(* Logix 5000 project; controller Sucrose_Main Emulate 5570 rev 20.12; software revision 20.01; part 21 of 30 *)
(* tags used below, declared in another part *)
   CIPRemote : Area_Program;
   FV140501_AOI : QSI_Flow_Valve;   // FV-14-05-01 PRE FILTER TRAIN 1 SUPPLY VALVE
   FV140502_AOI : QSI_Flow_Valve;   // FV-14-05-02 FINAL FILTER TRAIN 1 SUPPLY VALVE
   FV140503_AOI : QSI_Flow_Valve;   // FV-14-05-03 HOT WATER LOW POINT DRAIN VALVE
   FV140601_AOI : QSI_Flow_Valve;   // FV-14-06-01 PRE FILTER TRAIN 2 SUPPLY VALVE
   FV140602_AOI : QSI_Flow_Valve;   // FV-14-06-02 FINAL FILTER TRAIN 2 SUPPLY VALVE
   FV150501_AOI : QSI_Flow_Valve;   // FV-15-05-01 DIVERT TO SCRAP OR TO DRAIN VALVE
   FV230500_AOI : QSI_Flow_Valve;   // FV-23-05-00 SUCROSE LOW POINT DRAIN VALVE
   FV230501_AOI : QSI_Flow_Valve;   // FV-23-05-01-O PRE FILTER TRAIN 1 INLET VALVE OPEN
   FV230502_AOI : QSI_Flow_Valve;   // FV-23-05-02 PRE FILTER TRAIN 1 INLET LOW POINT DRAIN VALVE
   FV230503_AOI : QSI_Flow_Valve;   // FV-23-05-03 PRE FILTER TRAIN 1 INLET LOW POINT DRAIN VALVE
   FV230504_AOI : QSI_Flow_Valve;   // FV-23-05-04 PRE FILTER TRAIN 1 OUTLET LOW POINT DRAIN VALVE
   FV230505_AOI : QSI_Flow_Valve;   // FV-23-05-05 PRE FILTER TRAIN 1 OUTLET LOW POINT DRAIN VALVE
   FV230506_AOI : QSI_Flow_Valve;   // FV-23-05-06-O PRE FILTER TRAIN 1 OUTLET VALVE OPEN
   FV230508_AOI : QSI_Flow_Valve;   // FV-23-05-08-O FINAL FILTER TRAIN 1 INLET VALVE OPEN
   FV230509_AOI : QSI_Flow_Valve;   // FV-23-05-09 FINAL FILTER TRAIN 1 INLET LOW POINT DRAIN VALVE
   FV230510_AOI : QSI_Flow_Valve;   // FV-23-05-10 FINAL FILTER TRAIN 1 INLET LOW POINT DRAIN VALVE
   FV230511_AOI : QSI_Flow_Valve;   // FV-23-05-11 FINAL FILTER TRAIN 1 OUTLET LOW POINT DRAIN VALVE
   FV230512_AOI : QSI_Flow_Valve;   // FV-23-05-12 FINAL FILTER TRAIN 1 OUTLET LOW POINT DRAIN VALVE
   FV230513_AOI : QSI_Flow_Valve;   // FV-23-05-13-O FINAL FILTER TRAIN 1 OUTLET VALVE OPEN
   FV230601_AOI : QSI_Flow_Valve;   // FV-23-06-01-O PRE FILTER TRAIN 2 INLET VALVE OPEN
   FV230602_AOI : QSI_Flow_Valve;   // FV-23-06-02 PRE FILTER TRAIN 2 INLET LOW POINT DRAIN VALVE
   FV230603_AOI : QSI_Flow_Valve;   // FV-23-06-03 PRE FILTER TRAIN 2 INLET LOW POINT DRAIN VALVE
   FV230604_AOI : QSI_Flow_Valve;   // FV-23-06-04 PRE FILTER TRAIN 2 OUTLET LOW POINT DRAIN VALVE
   FV230605_AOI : QSI_Flow_Valve;   // FV-23-06-05 PRE FILTER TRAIN 2 OUTLET LOW POINT DRAIN VALVE
   FV230606_AOI : QSI_Flow_Valve;   // FV-23-06-06-O PRE FILTER TRAIN 2 OUTLET VALVE OPEN
   FV230607_AOI : QSI_Flow_Valve;   // FV-23-06-07 LOW POINT DRAIN VALVE
   FV230608_AOI : QSI_Flow_Valve;   // FV-23-06-08-O FINAL FILTER TRAIN 2 INLET VALVE OPEN
   FV230609_AOI : QSI_Flow_Valve;   // FV-23-06-09 FINAL FILTER TRAIN 2 INLET LOW POINT DRAIN VALVE
   FV230610_AOI : QSI_Flow_Valve;   // FV-23-06-10 FINAL FILTER TRAIN 2 INLET LOW POINT DRAIN VALVE
   FV230611_AOI : QSI_Flow_Valve;   // FV-23-06-11 FINAL FILTER TRAIN 2 OUTLET LOW POINT DRAIN VALVE
   FV230612_AOI : QSI_Flow_Valve;   // FV-23-06-12 FINAL FILTER TRAIN 2 OUTLET LOW POINT DRAIN VALVE
   FV230613_AOI : QSI_Flow_Valve;   // FV-23-06-13-O FINAL FILTER TRAIN 2 OUTLET VALVE OPEN
   ONESHOTBITS : INT[10];
   Rung_Comment : BOOL;
   SECURITY : User_Login;
   SucroseCIP_FILTRATION_REMOTE : CIP_REMOTE;
   SucroseCIP_RUNNING : BOOL;
   SucroseCIP_TK230101_REMOTE : CIP_REMOTE;
   SucroseCIP_TK230201_REMOTE : CIP_REMOTE;
   SucroseCIP_TK230301_REMOTE : CIP_REMOTE;
   SucroseFiltration : Area_Program;
(* Master_Main, continued *)

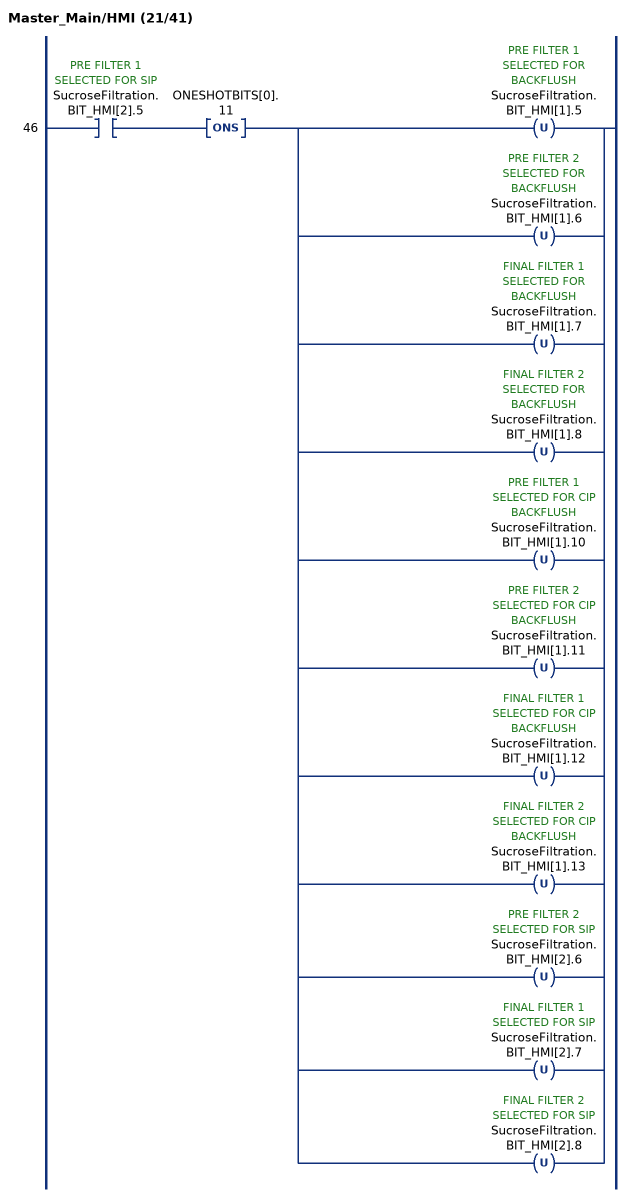
   46: XIC(SucroseFiltration.BIT_HMI[2].5)ONS(ONESHOTBITS[0].11)[OTU(SucroseFiltration.BIT_HMI[1].5) ,OTU(SucroseFiltration.BIT_HMI[1].6) ,OTU(SucroseFiltration.BIT_HMI[1].7) ,OTU(SucroseFiltration.BIT_HMI[1].8) ,OTU(SucroseFiltration.BIT_HMI[1].10) ,OTU(SucroseFiltration.BIT_HMI[1].11) ,OTU(SucroseFiltration.BIT_HMI[1].12) ,OTU(SucroseFiltration.BIT_HMI[1].13) ,OTU(SucroseFiltration.BIT_HMI[2].6) ,OTU(SucroseFiltration.BIT_HMI[2].7) ,OTU(SucroseFiltration.BIT_HMI[2].8) ];
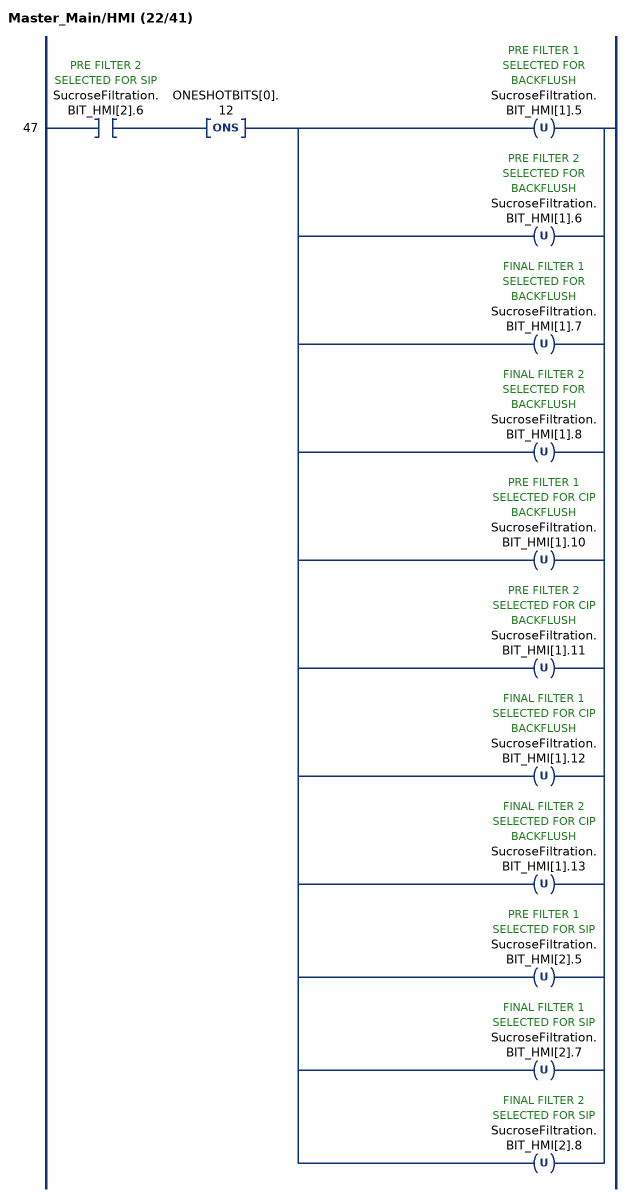
   47: XIC(SucroseFiltration.BIT_HMI[2].6)ONS(ONESHOTBITS[0].12)[OTU(SucroseFiltration.BIT_HMI[1].5) ,OTU(SucroseFiltration.BIT_HMI[1].6) ,OTU(SucroseFiltration.BIT_HMI[1].7) ,OTU(SucroseFiltration.BIT_HMI[1].8) ,OTU(SucroseFiltration.BIT_HMI[1].10) ,OTU(SucroseFiltration.BIT_HMI[1].11) ,OTU(SucroseFiltration.BIT_HMI[1].12) ,OTU(SucroseFiltration.BIT_HMI[1].13) ,OTU(SucroseFiltration.BIT_HMI[2].5) ,OTU(SucroseFiltration.BIT_HMI[2].7) ,OTU(SucroseFiltration.BIT_HMI[2].8) ];
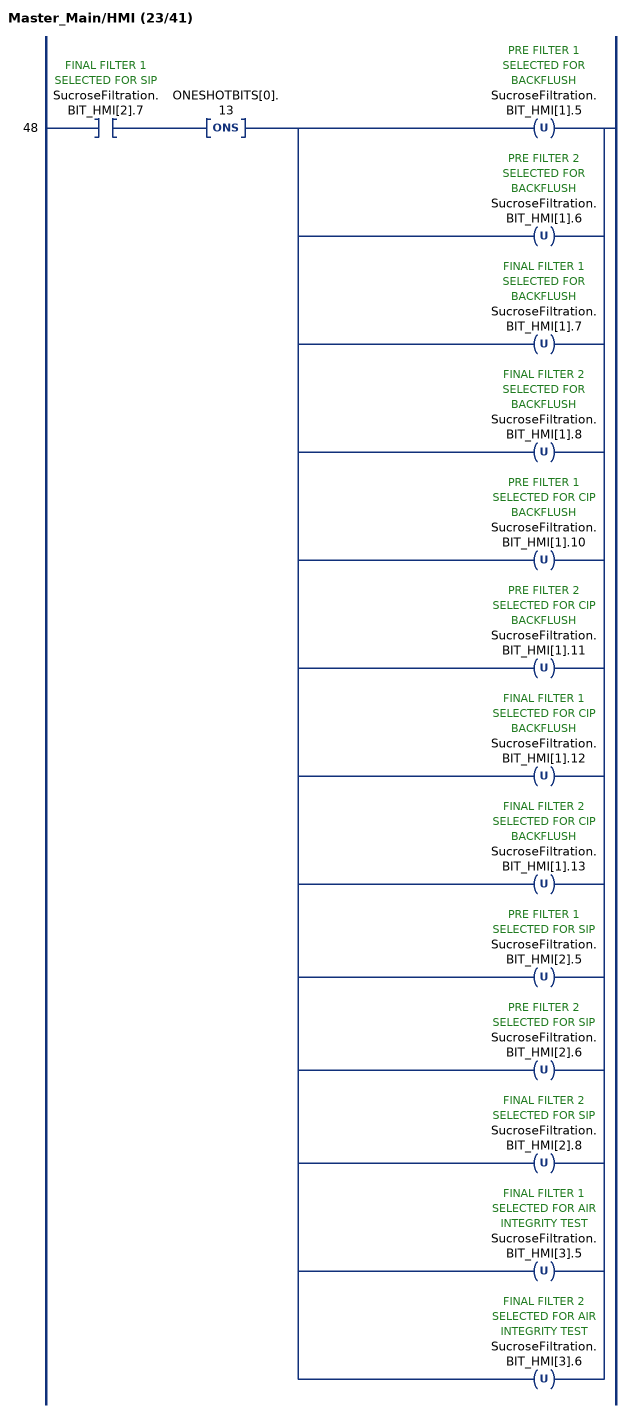
   48: XIC(SucroseFiltration.BIT_HMI[2].7)ONS(ONESHOTBITS[0].13)[OTU(SucroseFiltration.BIT_HMI[1].5) ,OTU(SucroseFiltration.BIT_HMI[1].6) ,OTU(SucroseFiltration.BIT_HMI[1].7) ,OTU(SucroseFiltration.BIT_HMI[1].8) ,OTU(SucroseFiltration.BIT_HMI[1].10) ,OTU(SucroseFiltration.BIT_HMI[1].11) ,OTU(SucroseFiltration.BIT_HMI[1].12) ,OTU(SucroseFiltration.BIT_HMI[1].13) ,OTU(SucroseFiltration.BIT_HMI[2].5) ,OTU(SucroseFiltration.BIT_HMI[2].6) ,OTU(SucroseFiltration.BIT_HMI[2].8) ,OTU(SucroseFiltration.BIT_HMI[3].5) ,OTU(SucroseFiltration.BIT_HMI[3].6) ];
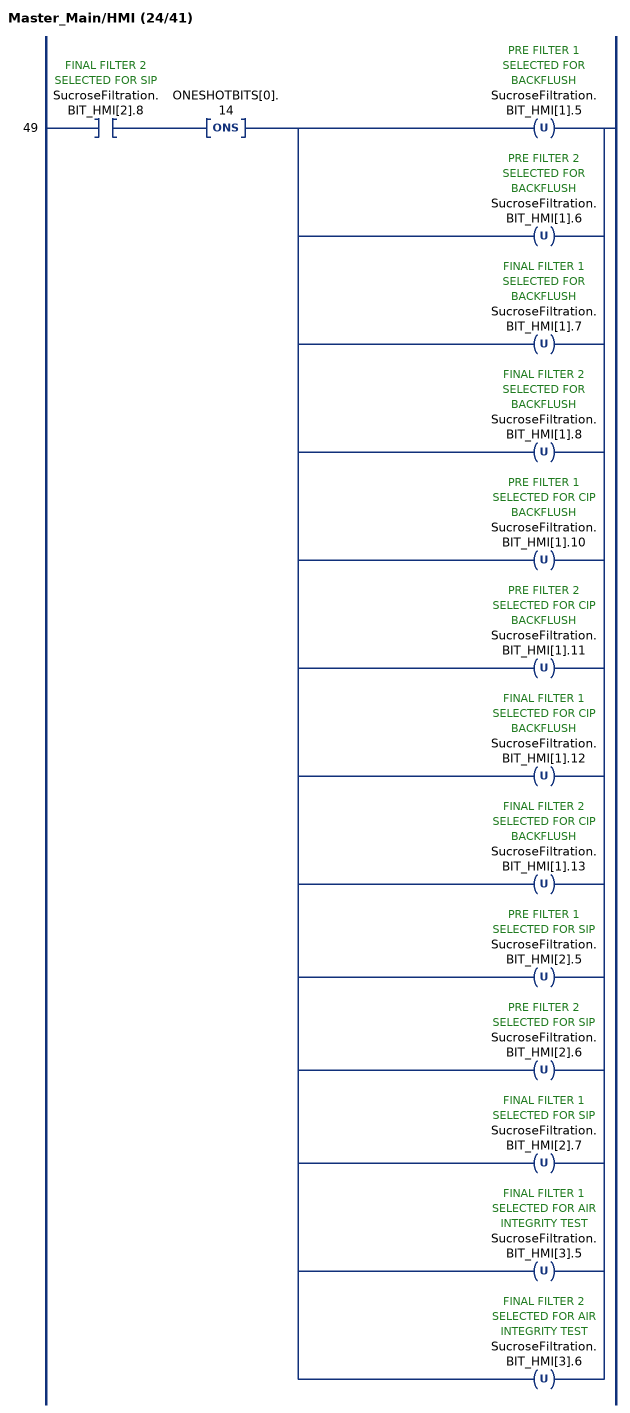
   49: XIC(SucroseFiltration.BIT_HMI[2].8)ONS(ONESHOTBITS[0].14)[OTU(SucroseFiltration.BIT_HMI[1].5) ,OTU(SucroseFiltration.BIT_HMI[1].6) ,OTU(SucroseFiltration.BIT_HMI[1].7) ,OTU(SucroseFiltration.BIT_HMI[1].8) ,OTU(SucroseFiltration.BIT_HMI[1].10) ,OTU(SucroseFiltration.BIT_HMI[1].11) ,OTU(SucroseFiltration.BIT_HMI[1].12) ,OTU(SucroseFiltration.BIT_HMI[1].13) ,OTU(SucroseFiltration.BIT_HMI[2].5) ,OTU(SucroseFiltration.BIT_HMI[2].6) ,OTU(SucroseFiltration.BIT_HMI[2].7) ,OTU(SucroseFiltration.BIT_HMI[3].5) ,OTU(SucroseFiltration.BIT_HMI[3].6) ];
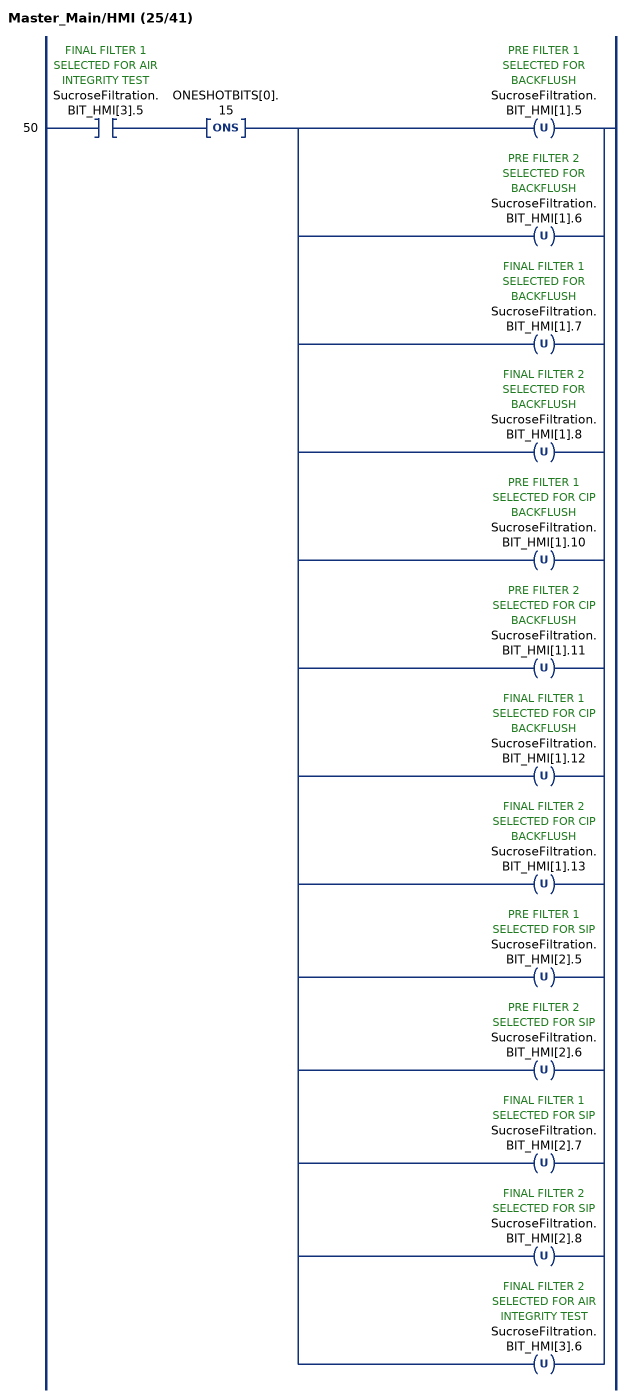
   50: XIC(SucroseFiltration.BIT_HMI[3].5)ONS(ONESHOTBITS[0].15)[OTU(SucroseFiltration.BIT_HMI[1].5) ,OTU(SucroseFiltration.BIT_HMI[1].6) ,OTU(SucroseFiltration.BIT_HMI[1].7) ,OTU(SucroseFiltration.BIT_HMI[1].8) ,OTU(SucroseFiltration.BIT_HMI[1].10) ,OTU(SucroseFiltration.BIT_HMI[1].11) ,OTU(SucroseFiltration.BIT_HMI[1].12) ,OTU(SucroseFiltration.BIT_HMI[1].13) ,OTU(SucroseFiltration.BIT_HMI[2].5) ,OTU(SucroseFiltration.BIT_HMI[2].6) ,OTU(SucroseFiltration.BIT_HMI[2].7) ,OTU(SucroseFiltration.BIT_HMI[2].8) ,OTU(SucroseFiltration.BIT_HMI[3].6) ];
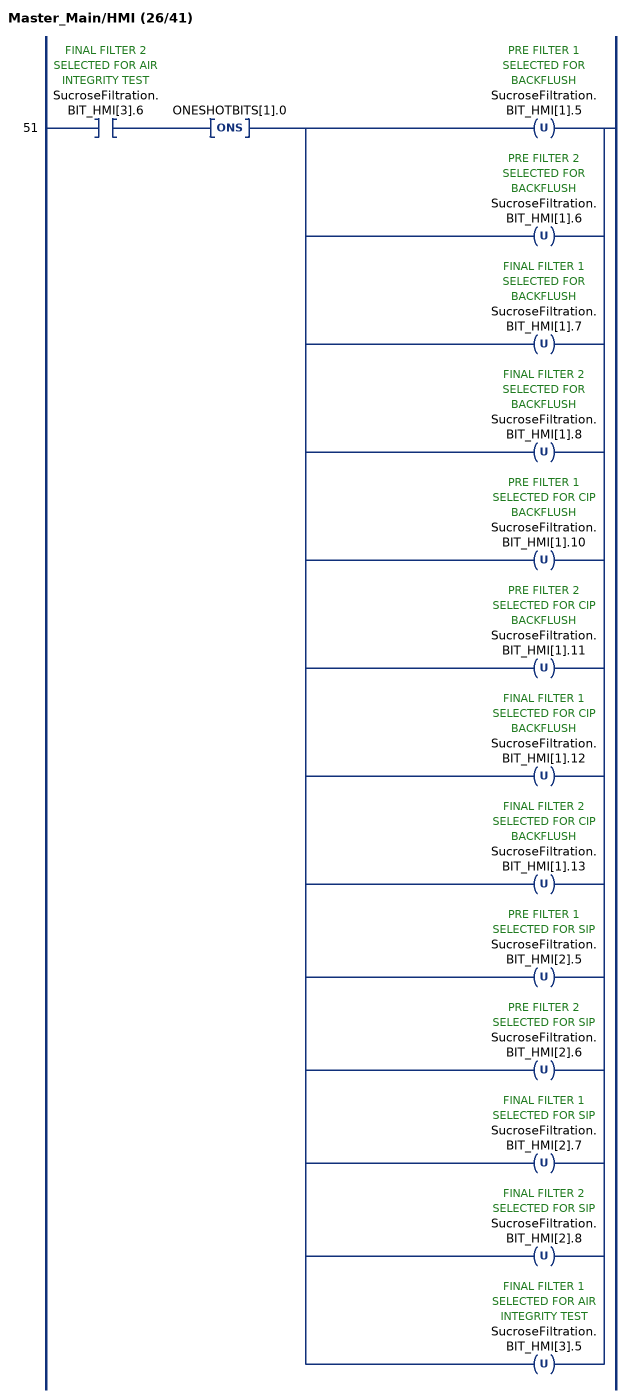
   51: XIC(SucroseFiltration.BIT_HMI[3].6)ONS(ONESHOTBITS[1].0)[OTU(SucroseFiltration.BIT_HMI[1].5) ,OTU(SucroseFiltration.BIT_HMI[1].6) ,OTU(SucroseFiltration.BIT_HMI[1].7) ,OTU(SucroseFiltration.BIT_HMI[1].8) ,OTU(SucroseFiltration.BIT_HMI[1].10) ,OTU(SucroseFiltration.BIT_HMI[1].11) ,OTU(SucroseFiltration.BIT_HMI[1].12) ,OTU(SucroseFiltration.BIT_HMI[1].13) ,OTU(SucroseFiltration.BIT_HMI[2].5) ,OTU(SucroseFiltration.BIT_HMI[2].6) ,OTU(SucroseFiltration.BIT_HMI[2].7) ,OTU(SucroseFiltration.BIT_HMI[2].8) ,OTU(SucroseFiltration.BIT_HMI[3].5) ];
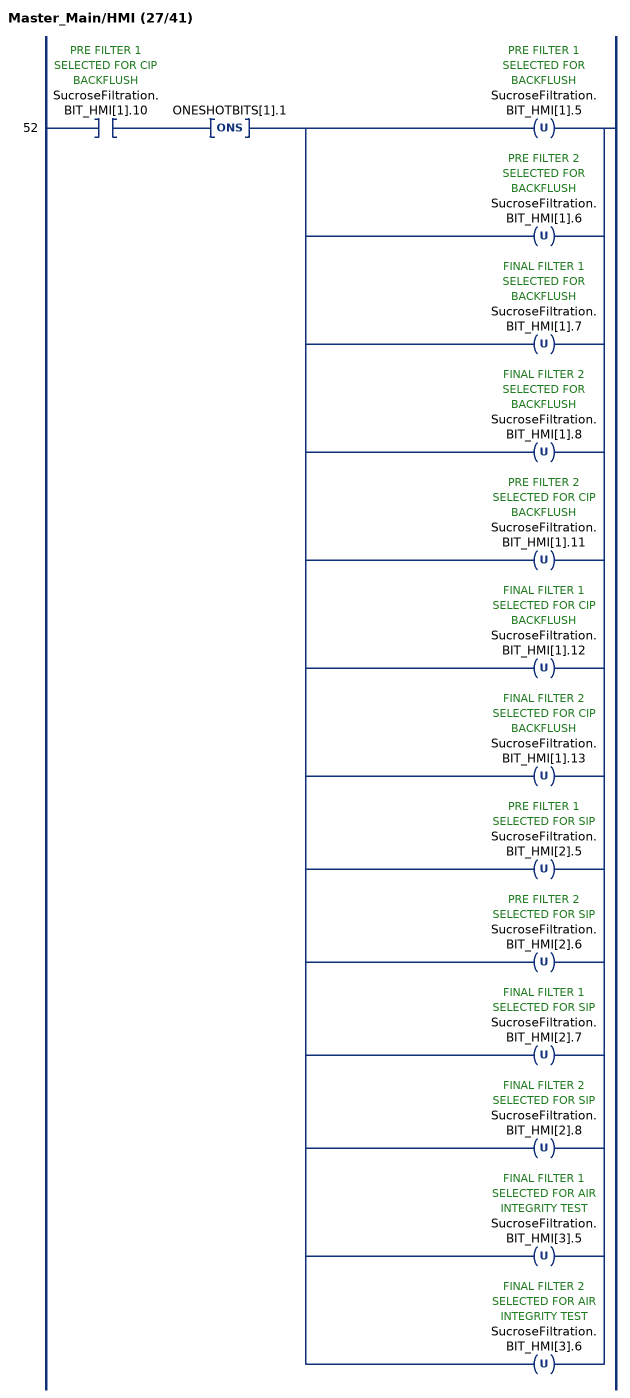
   52: XIC(SucroseFiltration.BIT_HMI[1].10)ONS(ONESHOTBITS[1].1)[OTU(SucroseFiltration.BIT_HMI[1].5) ,OTU(SucroseFiltration.BIT_HMI[1].6) ,OTU(SucroseFiltration.BIT_HMI[1].7) ,OTU(SucroseFiltration.BIT_HMI[1].8) ,OTU(SucroseFiltration.BIT_HMI[1].11) ,OTU(SucroseFiltration.BIT_HMI[1].12) ,OTU(SucroseFiltration.BIT_HMI[1].13) ,OTU(SucroseFiltration.BIT_HMI[2].5) ,OTU(SucroseFiltration.BIT_HMI[2].6) ,OTU(SucroseFiltration.BIT_HMI[2].7) ,OTU(SucroseFiltration.BIT_HMI[2].8) ,OTU(SucroseFiltration.BIT_HMI[3].5) ,OTU(SucroseFiltration.BIT_HMI[3].6) ];
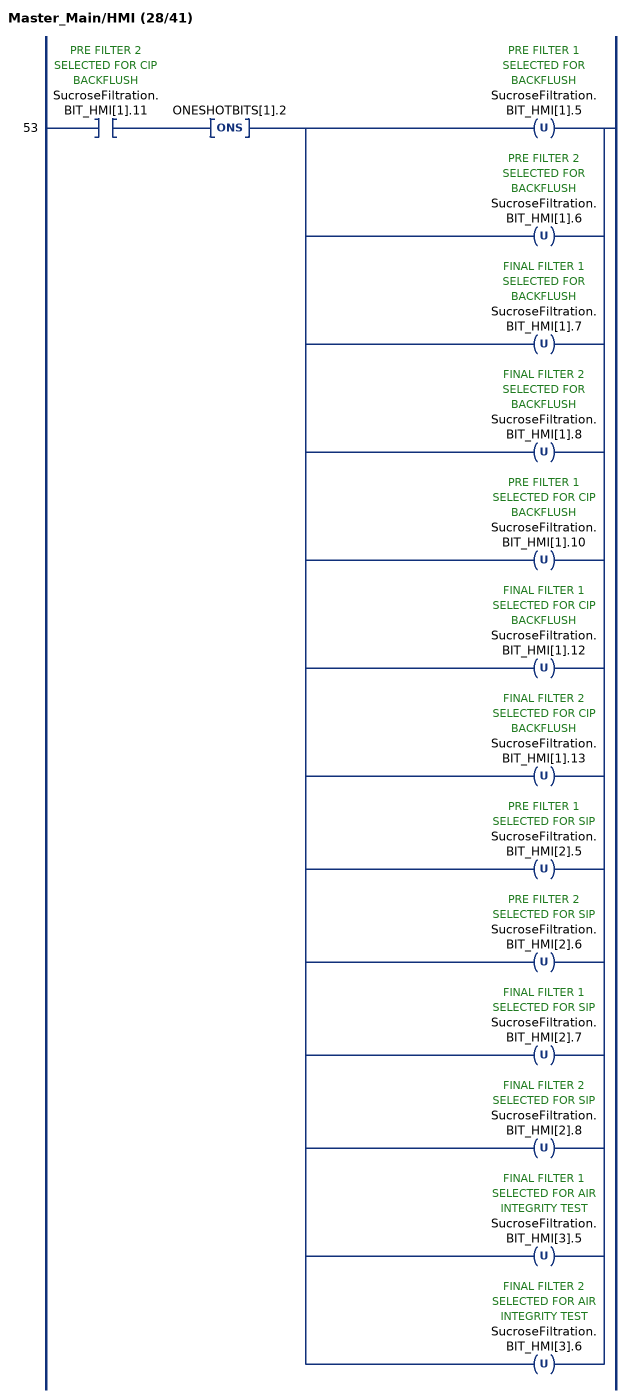
   53: XIC(SucroseFiltration.BIT_HMI[1].11)ONS(ONESHOTBITS[1].2)[OTU(SucroseFiltration.BIT_HMI[1].5) ,OTU(SucroseFiltration.BIT_HMI[1].6) ,OTU(SucroseFiltration.BIT_HMI[1].7) ,OTU(SucroseFiltration.BIT_HMI[1].8) ,OTU(SucroseFiltration.BIT_HMI[1].10) ,OTU(SucroseFiltration.BIT_HMI[1].12) ,OTU(SucroseFiltration.BIT_HMI[1].13) ,OTU(SucroseFiltration.BIT_HMI[2].5) ,OTU(SucroseFiltration.BIT_HMI[2].6) ,OTU(SucroseFiltration.BIT_HMI[2].7) ,OTU(SucroseFiltration.BIT_HMI[2].8) ,OTU(SucroseFiltration.BIT_HMI[3].5) ,OTU(SucroseFiltration.BIT_HMI[3].6) ];
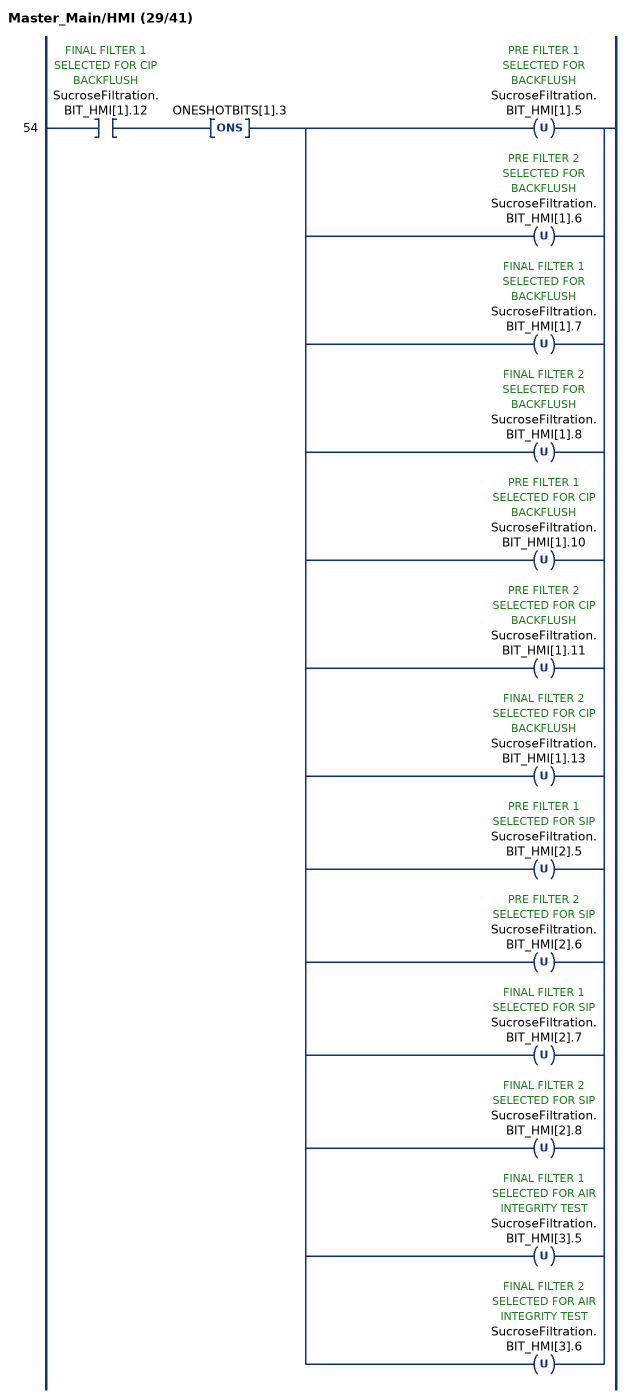
   54: XIC(SucroseFiltration.BIT_HMI[1].12)ONS(ONESHOTBITS[1].3)[OTU(SucroseFiltration.BIT_HMI[1].5) ,OTU(SucroseFiltration.BIT_HMI[1].6) ,OTU(SucroseFiltration.BIT_HMI[1].7) ,OTU(SucroseFiltration.BIT_HMI[1].8) ,OTU(SucroseFiltration.BIT_HMI[1].10) ,OTU(SucroseFiltration.BIT_HMI[1].11) ,OTU(SucroseFiltration.BIT_HMI[1].13) ,OTU(SucroseFiltration.BIT_HMI[2].5) ,OTU(SucroseFiltration.BIT_HMI[2].6) ,OTU(SucroseFiltration.BIT_HMI[2].7) ,OTU(SucroseFiltration.BIT_HMI[2].8) ,OTU(SucroseFiltration.BIT_HMI[3].5) ,OTU(SucroseFiltration.BIT_HMI[3].6) ];
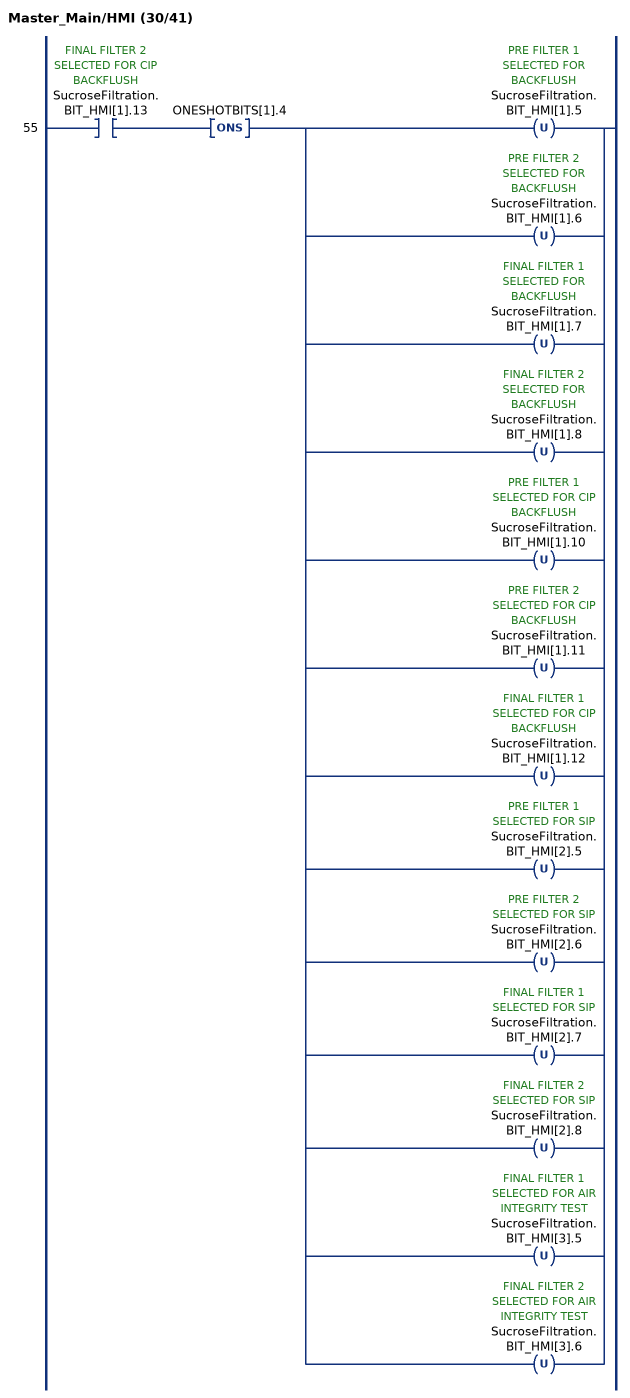
   55: XIC(SucroseFiltration.BIT_HMI[1].13)ONS(ONESHOTBITS[1].4)[OTU(SucroseFiltration.BIT_HMI[1].5) ,OTU(SucroseFiltration.BIT_HMI[1].6) ,OTU(SucroseFiltration.BIT_HMI[1].7) ,OTU(SucroseFiltration.BIT_HMI[1].8) ,OTU(SucroseFiltration.BIT_HMI[1].10) ,OTU(SucroseFiltration.BIT_HMI[1].11) ,OTU(SucroseFiltration.BIT_HMI[1].12) ,OTU(SucroseFiltration.BIT_HMI[2].5) ,OTU(SucroseFiltration.BIT_HMI[2].6) ,OTU(SucroseFiltration.BIT_HMI[2].7) ,OTU(SucroseFiltration.BIT_HMI[2].8) ,OTU(SucroseFiltration.BIT_HMI[3].5) ,OTU(SucroseFiltration.BIT_HMI[3].6) ];
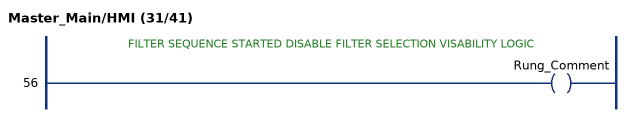
   // FILTER SEQUENCE STARTED DISABLE FILTER SELECTION VISABILITY LOGIC
   56: OTE(Rung_Comment);
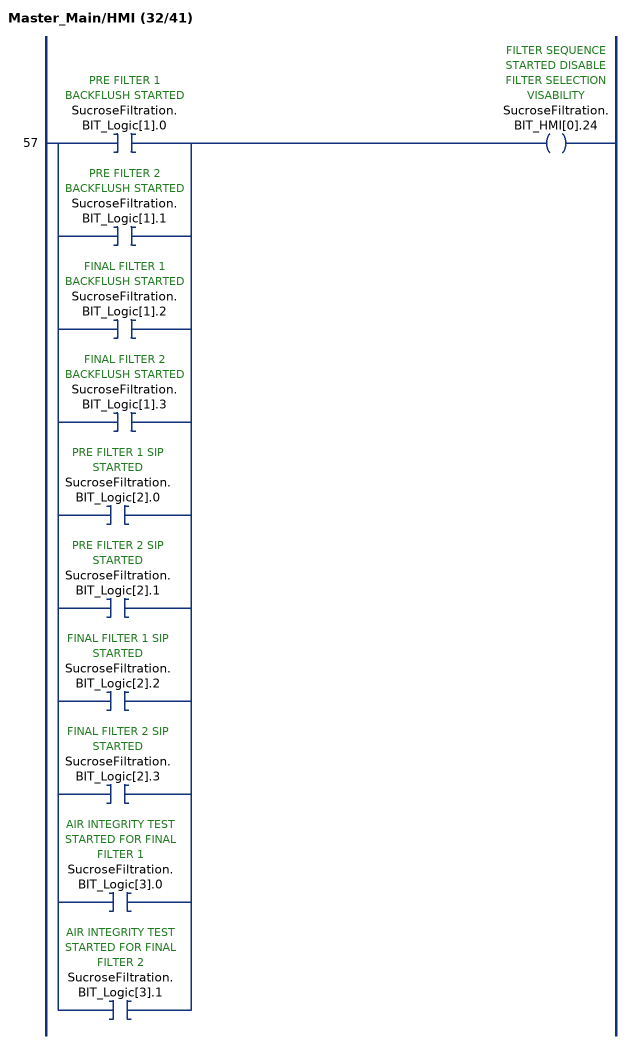
   57: [XIC(SucroseFiltration.BIT_Logic[1].0) ,XIC(SucroseFiltration.BIT_Logic[1].1) ,XIC(SucroseFiltration.BIT_Logic[1].2) ,XIC(SucroseFiltration.BIT_Logic[1].3) ,XIC(SucroseFiltration.BIT_Logic[2].0) ,XIC(SucroseFiltration.BIT_Logic[2].1) ,XIC(SucroseFiltration.BIT_Logic[2].2) ,XIC(SucroseFiltration.BIT_Logic[2].3) ,XIC(SucroseFiltration.BIT_Logic[3].0) ,XIC(SucroseFiltration.BIT_Logic[3].1) ]OTE(SucroseFiltration.BIT_HMI[0].24);
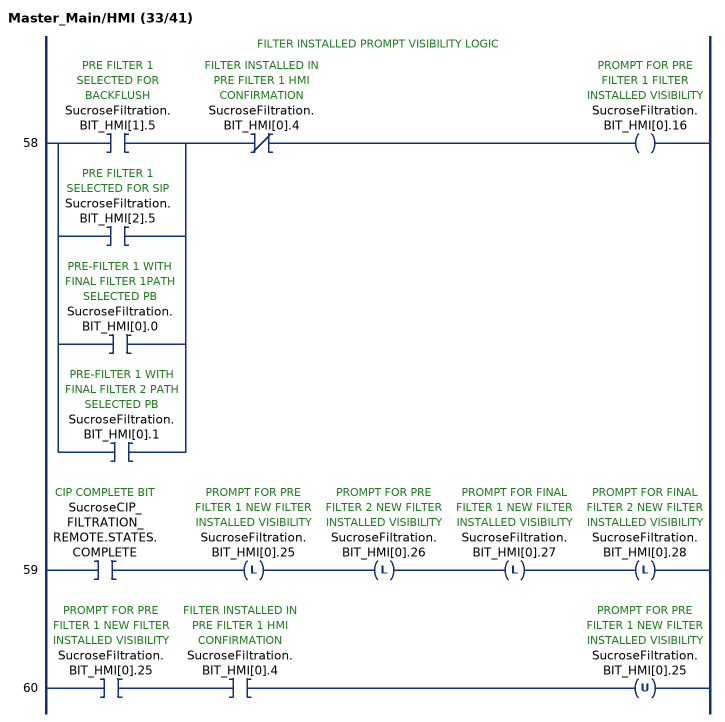
   // FILTER INSTALLED PROMPT VISIBILITY LOGIC
   58: [XIC(SucroseFiltration.BIT_HMI[1].5) ,XIC(SucroseFiltration.BIT_HMI[2].5) ,XIC(SucroseFiltration.BIT_HMI[0].0) ,XIC(SucroseFiltration.BIT_HMI[0].1) ]XIO(SucroseFiltration.BIT_HMI[0].4)OTE(SucroseFiltration.BIT_HMI[0].16);
   59: XIC(SucroseCIP_FILTRATION_REMOTE.STATES.COMPLETE)OTL(SucroseFiltration.BIT_HMI[0].25)OTL(SucroseFiltration.BIT_HMI[0].26)OTL(SucroseFiltration.BIT_HMI[0].27)OTL(SucroseFiltration.BIT_HMI[0].28);
   60: XIC(SucroseFiltration.BIT_HMI[0].25)XIC(SucroseFiltration.BIT_HMI[0].4)OTU(SucroseFiltration.BIT_HMI[0].25);
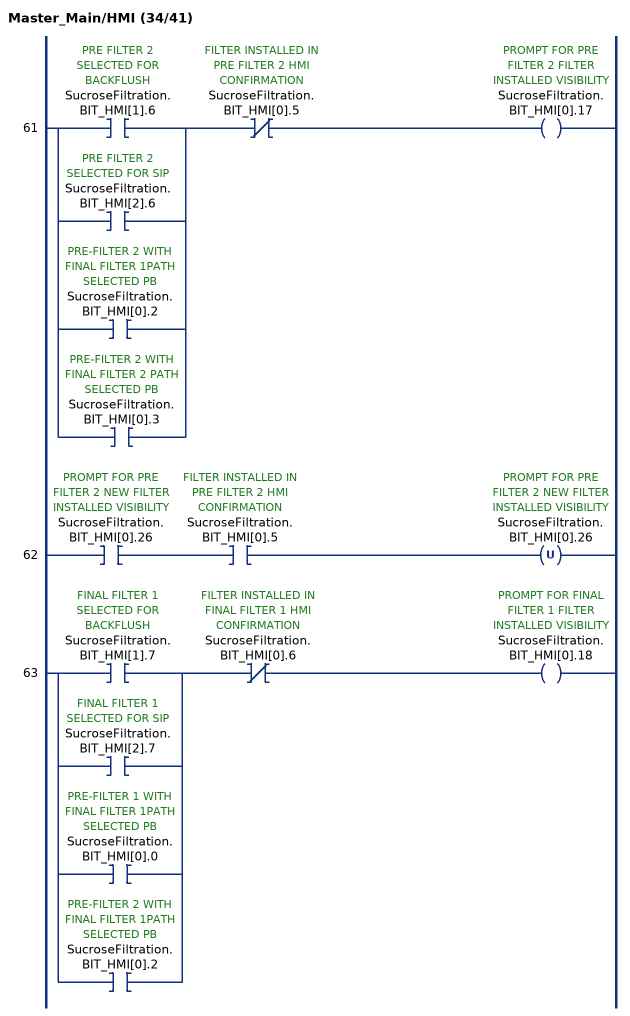
   61: [XIC(SucroseFiltration.BIT_HMI[1].6) ,XIC(SucroseFiltration.BIT_HMI[2].6) ,XIC(SucroseFiltration.BIT_HMI[0].2) ,XIC(SucroseFiltration.BIT_HMI[0].3) ]XIO(SucroseFiltration.BIT_HMI[0].5)OTE(SucroseFiltration.BIT_HMI[0].17);
   62: XIC(SucroseFiltration.BIT_HMI[0].26)XIC(SucroseFiltration.BIT_HMI[0].5)OTU(SucroseFiltration.BIT_HMI[0].26);
   63: [XIC(SucroseFiltration.BIT_HMI[1].7) ,XIC(SucroseFiltration.BIT_HMI[2].7) ,XIC(SucroseFiltration.BIT_HMI[0].0) ,XIC(SucroseFiltration.BIT_HMI[0].2) ]XIO(SucroseFiltration.BIT_HMI[0].6)OTE(SucroseFiltration.BIT_HMI[0].18);
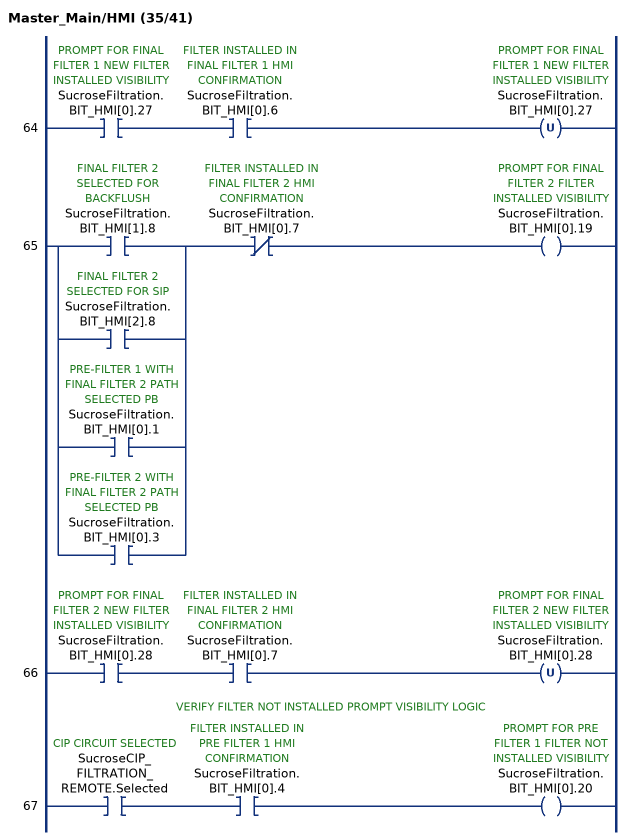
   64: XIC(SucroseFiltration.BIT_HMI[0].27)XIC(SucroseFiltration.BIT_HMI[0].6)OTU(SucroseFiltration.BIT_HMI[0].27);
   65: [XIC(SucroseFiltration.BIT_HMI[1].8) ,XIC(SucroseFiltration.BIT_HMI[2].8) ,XIC(SucroseFiltration.BIT_HMI[0].1) ,XIC(SucroseFiltration.BIT_HMI[0].3) ]XIO(SucroseFiltration.BIT_HMI[0].7)OTE(SucroseFiltration.BIT_HMI[0].19);
   66: XIC(SucroseFiltration.BIT_HMI[0].28)XIC(SucroseFiltration.BIT_HMI[0].7)OTU(SucroseFiltration.BIT_HMI[0].28);
   // VERIFY FILTER NOT INSTALLED PROMPT VISIBILITY LOGIC
   67: XIC(SucroseCIP_FILTRATION_REMOTE.Selected)XIC(SucroseFiltration.BIT_HMI[0].4)OTE(SucroseFiltration.BIT_HMI[0].20);
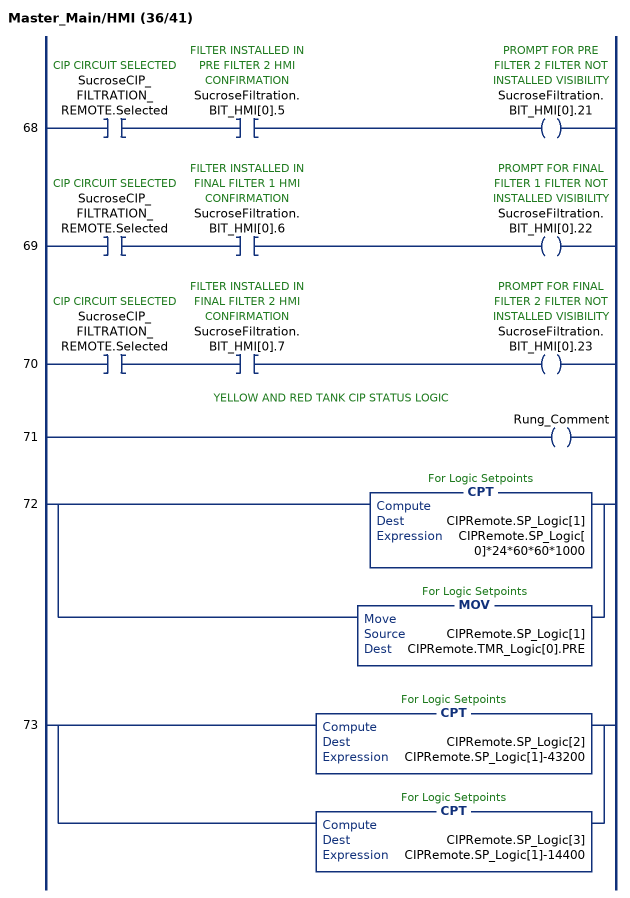
   68: XIC(SucroseCIP_FILTRATION_REMOTE.Selected)XIC(SucroseFiltration.BIT_HMI[0].5)OTE(SucroseFiltration.BIT_HMI[0].21);
   69: XIC(SucroseCIP_FILTRATION_REMOTE.Selected)XIC(SucroseFiltration.BIT_HMI[0].6)OTE(SucroseFiltration.BIT_HMI[0].22);
   70: XIC(SucroseCIP_FILTRATION_REMOTE.Selected)XIC(SucroseFiltration.BIT_HMI[0].7)OTE(SucroseFiltration.BIT_HMI[0].23);
   // YELLOW AND RED TANK CIP STATUS LOGIC
   71: OTE(Rung_Comment);
   72: [CPT(CIPRemote.SP_Logic[1],CIPRemote.SP_Logic[0]*24*60*60*1000) ,MOV(CIPRemote.SP_Logic[1],CIPRemote.TMR_Logic[0].PRE) ];
   73: [CPT(CIPRemote.SP_Logic[2],CIPRemote.SP_Logic[1]-43200) ,CPT(CIPRemote.SP_Logic[3],CIPRemote.SP_Logic[1]-14400) ];
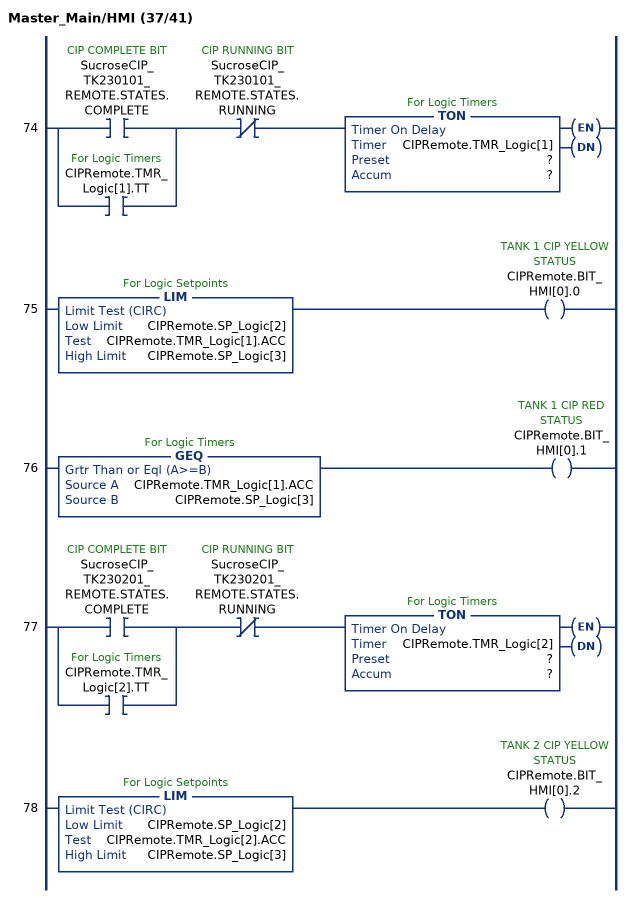
   74: [XIC(SucroseCIP_TK230101_REMOTE.STATES.COMPLETE) ,XIC(CIPRemote.TMR_Logic[1].TT) ]XIO(SucroseCIP_TK230101_REMOTE.STATES.RUNNING)TON(CIPRemote.TMR_Logic[1],?,?);
   75: LIM(CIPRemote.SP_Logic[2],CIPRemote.TMR_Logic[1].ACC,CIPRemote.SP_Logic[3])OTE(CIPRemote.BIT_HMI[0].0);
   76: GEQ(CIPRemote.TMR_Logic[1].ACC,CIPRemote.SP_Logic[3])OTE(CIPRemote.BIT_HMI[0].1);
   77: [XIC(SucroseCIP_TK230201_REMOTE.STATES.COMPLETE) ,XIC(CIPRemote.TMR_Logic[2].TT) ]XIO(SucroseCIP_TK230201_REMOTE.STATES.RUNNING)TON(CIPRemote.TMR_Logic[2],?,?);
   78: LIM(CIPRemote.SP_Logic[2],CIPRemote.TMR_Logic[2].ACC,CIPRemote.SP_Logic[3])OTE(CIPRemote.BIT_HMI[0].2);
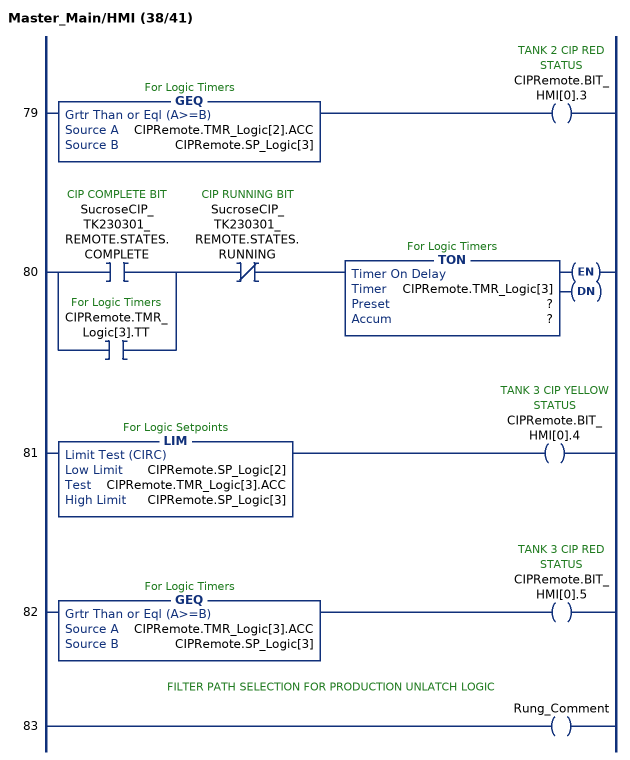
   79: GEQ(CIPRemote.TMR_Logic[2].ACC,CIPRemote.SP_Logic[3])OTE(CIPRemote.BIT_HMI[0].3);
   80: [XIC(SucroseCIP_TK230301_REMOTE.STATES.COMPLETE) ,XIC(CIPRemote.TMR_Logic[3].TT) ]XIO(SucroseCIP_TK230301_REMOTE.STATES.RUNNING)TON(CIPRemote.TMR_Logic[3],?,?);
   81: LIM(CIPRemote.SP_Logic[2],CIPRemote.TMR_Logic[3].ACC,CIPRemote.SP_Logic[3])OTE(CIPRemote.BIT_HMI[0].4);
   82: GEQ(CIPRemote.TMR_Logic[3].ACC,CIPRemote.SP_Logic[3])OTE(CIPRemote.BIT_HMI[0].5);
   // FILTER PATH SELECTION FOR PRODUCTION UNLATCH LOGIC
   83: OTE(Rung_Comment);
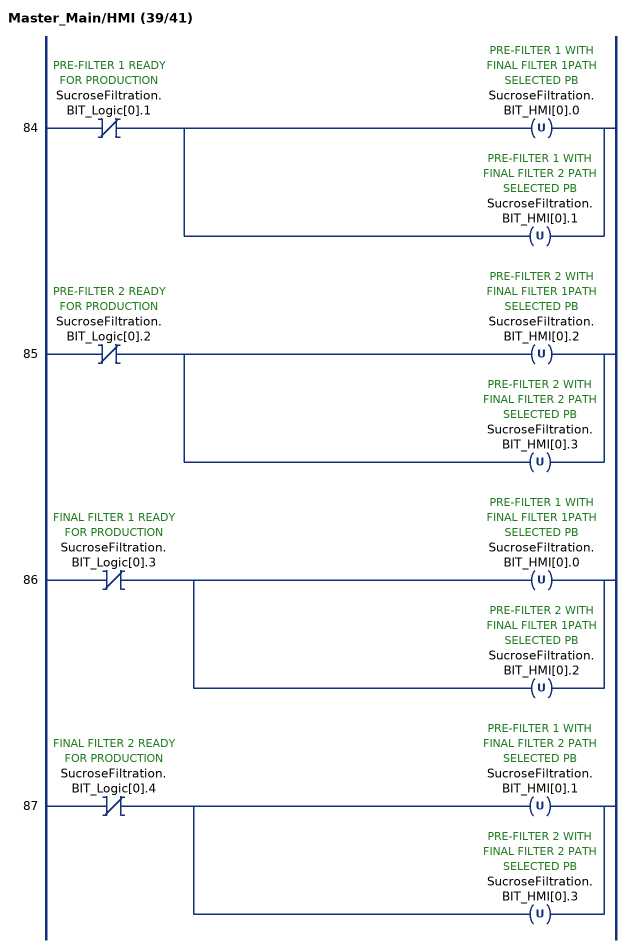
   84: XIO(SucroseFiltration.BIT_Logic[0].1)[OTU(SucroseFiltration.BIT_HMI[0].0) ,OTU(SucroseFiltration.BIT_HMI[0].1) ];
   85: XIO(SucroseFiltration.BIT_Logic[0].2)[OTU(SucroseFiltration.BIT_HMI[0].2) ,OTU(SucroseFiltration.BIT_HMI[0].3) ];
   86: XIO(SucroseFiltration.BIT_Logic[0].3)[OTU(SucroseFiltration.BIT_HMI[0].0) ,OTU(SucroseFiltration.BIT_HMI[0].2) ];
   87: XIO(SucroseFiltration.BIT_Logic[0].4)[OTU(SucroseFiltration.BIT_HMI[0].1) ,OTU(SucroseFiltration.BIT_HMI[0].3) ];
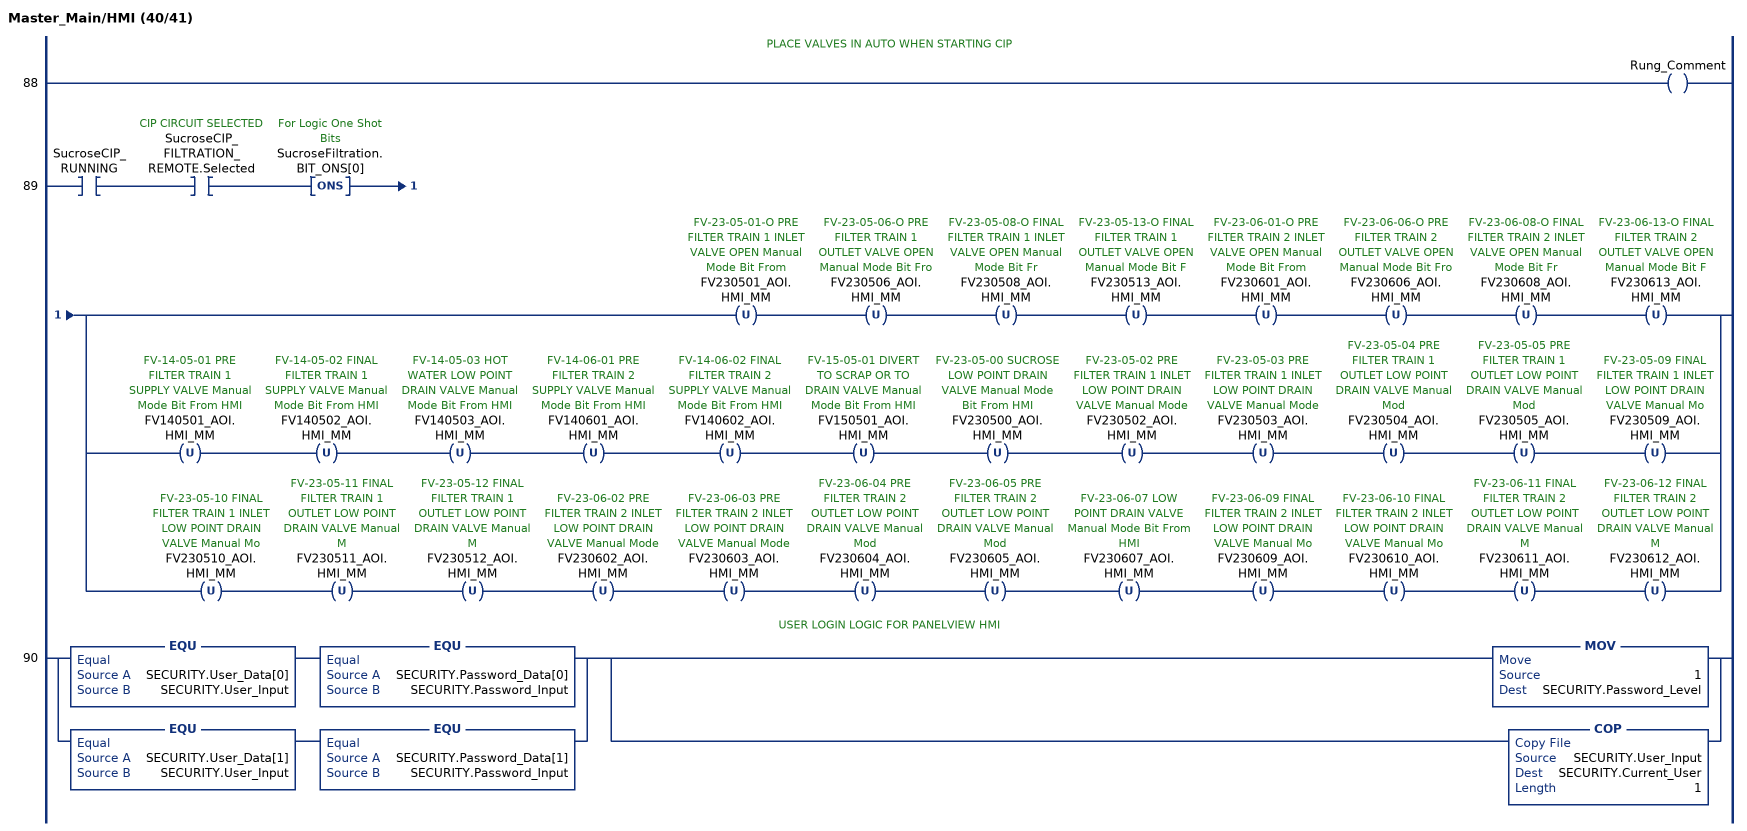
   // PLACE VALVES IN AUTO WHEN STARTING CIP
   88: OTE(Rung_Comment);
   89: XIC(SucroseCIP_RUNNING)XIC(SucroseCIP_FILTRATION_REMOTE.Selected)ONS(SucroseFiltration.BIT_ONS[0])[OTU(FV230501_AOI.HMI_MM) OTU(FV230506_AOI.HMI_MM) OTU(FV230508_AOI.HMI_MM) OTU(FV230513_AOI.HMI_MM) OTU(FV230601_AOI.HMI_MM) OTU(FV230606_AOI.HMI_MM) OTU(FV230608_AOI.HMI_MM) OTU(FV230613_AOI.HMI_MM) ,OTU(FV140501_AOI.HMI_MM) OTU(FV140502_AOI.HMI_MM) OTU(FV140503_AOI.HMI_MM) OTU(FV140601_AOI.HMI_MM) OTU(FV140602_AOI.HMI_MM) OTU(FV150501_AOI.HMI_MM) OTU(FV230500_AOI.HMI_MM) OTU(FV230502_AOI.HMI_MM) OTU(FV230503_AOI.HMI_MM) OTU(FV230504_AOI.HMI_MM) OTU(FV230505_AOI.HMI_MM) OTU(FV230509_AOI.HMI_MM) ,OTU(FV230510_AOI.HMI_MM) OTU(FV230511_AOI.HMI_MM) OTU(FV230512_AOI.HMI_MM) OTU(FV230602_AOI.HMI_MM) OTU(FV230603_AOI.HMI_MM) OTU(FV230604_AOI.HMI_MM) OTU(FV230605_AOI.HMI_MM) OTU(FV230607_AOI.HMI_MM) OTU(FV230609_AOI.HMI_MM) OTU(FV230610_AOI.HMI_MM) OTU(FV230611_AOI.HMI_MM) OTU(FV230612_AOI.HMI_MM) ];
   // USER LOGIN LOGIC FOR PANELVIEW HMI
   90: [EQU(SECURITY.User_Data[0],SECURITY.User_Input) EQU(SECURITY.Password_Data[0],SECURITY.Password_Input) ,EQU(SECURITY.User_Data[1],SECURITY.User_Input) EQU(SECURITY.Password_Data[1],SECURITY.Password_Input) ][MOV(1,SECURITY.Password_Level) ,COP(SECURITY.User_Input,SECURITY.Current_User,1) ];
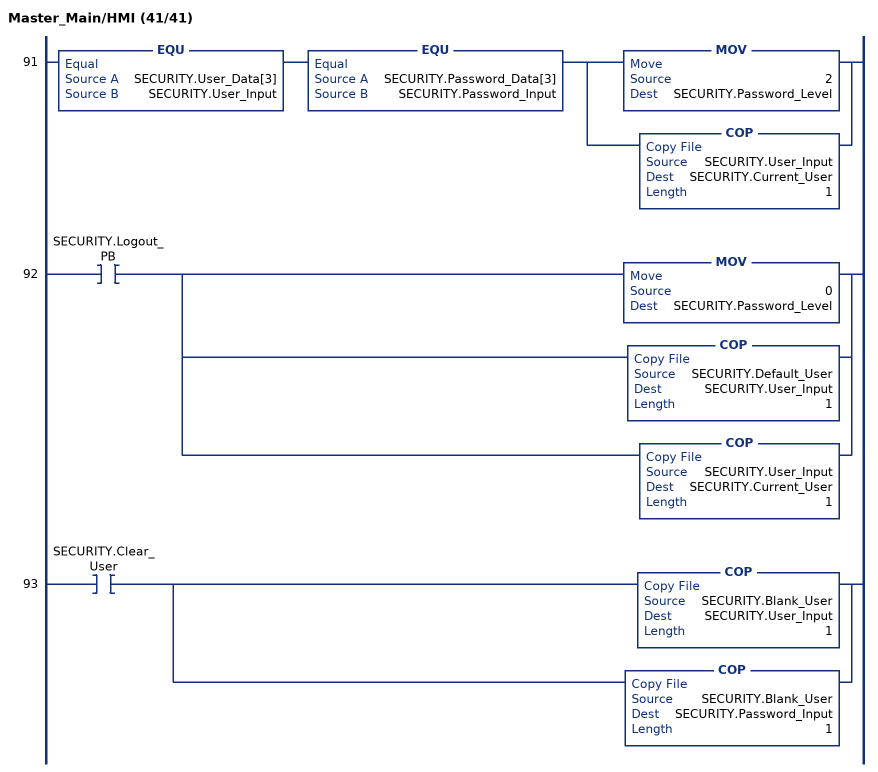
   91: EQU(SECURITY.User_Data[3],SECURITY.User_Input)EQU(SECURITY.Password_Data[3],SECURITY.Password_Input)[MOV(2,SECURITY.Password_Level) ,COP(SECURITY.User_Input,SECURITY.Current_User,1) ];
   92: XIC(SECURITY.Logout_PB)[MOV(0,SECURITY.Password_Level) ,COP(SECURITY.Default_User,SECURITY.User_Input,1) ,COP(SECURITY.User_Input,SECURITY.Current_User,1) ];
   93: XIC(SECURITY.Clear_User)[COP(SECURITY.Blank_User,SECURITY.User_Input,1) ,COP(SECURITY.Blank_User,SECURITY.Password_Input,1) ];
END_ROUTINE
